PROGRAM main
  VAR
    Start_PB : BOOL;
    Stop_PB : BOOL;
    Motor : BOOL;
    RunCmd : BOOL;
    TON0 : TON;
  END_VAR

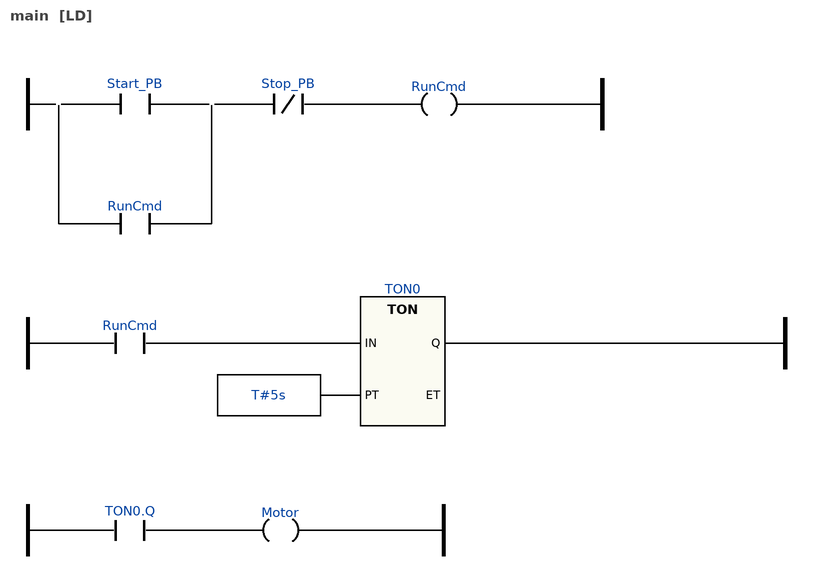
(* LD diagram, written out as Structured Text *)
RunCmd := (Start_PB OR RunCmd) AND NOT Stop_PB;
Motor := TON0.Q;
TON0(IN := RunCmd, PT := T#5s);
END_PROGRAM
